(* IEC 61131-3 sources: CodesysTest/export/UN00 - Sharp Bagger/EM01 - Bagger Head/CM04 - Bag Delivery/FB_SXBagDelivery.pou, 3 files *)

(* ---- FB_SXBagDelivery.pou.st ---- *)
(*#-#-#-#-#-#-#-#-#-#---Declaration---#-#-#-#-#-#-#-#-#-#-#-#-#*)

FUNCTION_BLOCK FINAL FB_SXBagDelivery EXTENDS FB_BaseComponent IMPLEMENTS IBagDelivery
VAR_INPUT
	simulateIO : BOOL;
	dryCycleEnable : BOOL;
	bagPresent : BOOL;
	printer : IPrinter;
	bagLength : REAL := 24.0;
	feedSpeed : REAL := 30.0;
	reverseSpeed : REAL := 3.0;
	printSpeed : REAL := 6.0;
	printOffset : REAL := 4.5;
	printLength : REAL := 6.0;
	maxReverseSetpoint : REAL := 3.0;
	sealOffset : REAL := 1.5;
	distanceFromSealBarToBagEdge : REAL := 3;
	distanceFromNipToBagEdge : REAL := 1.25;
	trapezoidalPercent : REAL := 0.1;
END_VAR
VAR_OUTPUT
	reverseFault : FB_Fault(name := Standard.CONCAT(_prefix,'Reverse Fault'));
	bagFailedToSeparate : FB_Fault(name := Standard.CONCAT(_prefix,'Failed To Separate'));
	noBagOverEye : FB_Fault(name := Standard.CONCAT(_prefix,'No Bag Over Photoeye'));
	motorFault : FB_Fault(name := CONCAT(_prefix, 'Film Feed Motor Fault'));
	motorCommFault : FB_Fault(name := CONCAT(_prefix, 'Film Feed Motor Comm Fault'));
END_VAR
VAR
	_feedAtPrintSpeed : BOOL;
	_feedBagOut : BOOL;
	_feedToPrintOffset : BOOL;
	_reverseToSeparate : BOOL;
	_bagFeedDone : BOOL;
	_bagSeparated : BOOL;
	_readyForPrint : BOOL;
	state : INT;
	nextState : INT;
	moveBagDeliveryTimeout : Standard.TON;
	MC_MoveBagDelivery : MC_MoveRelative;
	MC_HaltBagDelivery : MC_Halt;
	MC_ResetBagDelivery : MC_Reset;
	remainingLength : REAL;
	bagReversedToPrintOffset : BOOL;
	bagEdgePhotoeyeSim : FB_SimulatedFeedbackPhysicalInput(name := 'Bag Edge Photoeye Sim');
	printingNow : BOOL;
END_VAR
VAR_IN_OUT
	bagDeliveryMotor : Axis_REF;
END_VAR(*#-#-#-#-#-#-#-#-#-#---Implementation---#-#-#-#-#-#-#-#-#-#-#-#-#*)

SUPER^();

{region "Axis Setup"}
// Setup of Motion Commands for Bag Delivery motor axis
MC_MoveBagDelivery(Axis := bagDeliveryMotor);
MC_HaltBagDelivery(Axis := bagDeliveryMotor);
MC_ResetBagDelivery(Axis := bagDeliveryMotor);
{endregion}

IF MC_ResetBagDelivery.Execute THEN
	MC_ResetBagDelivery.Execute := FALSE;
END_IF

IF resetONS.Q THEN
	state := 100;
	nextState := 0;
	ClearStatus();
	IF bagDeliveryMotor.Error OR NOT bagDeliveryMotor.CommStatus THEN
		MC_ResetBagDelivery.Execute := TRUE;
	END_IF
END_IF

_ready := state = 0 AND bagDeliveryMotor.CommStatus AND NOT bagDeliveryMotor.Error;
IF bagDeliveryMotor.Error THEN
	motorFault.faultTrigger := TRUE;
ELSE
	motorFault.faultTrigger := FALSE;
END_IF

IF NOT bagDeliveryMotor.CommStatus THEN
	motorCommFault.faultTrigger := TRUE;
ELSE
	motorCommFault.faultTrigger := FALSE;
END_IF

IF trapezoidalPercent <= 0 THEN
	trapezoidalPercent := 0.1;
END_IF

CASE state OF
	0:		// Idle
			IF _feedBagOut THEN
				state := 10;
				_feedBagOut := FALSE;
				ClearStatus();
			END_IF

			IF _feedToPrintOffset THEN
				state := 20;
				_feedToPrintOffset := FALSE;
				ClearStatus();
			END_IF

			IF _reverseToSeparate THEN
				_bagSeparated := FALSE;
				state := 50;
				_reverseToSeparate := FALSE;
				ClearStatus();
			END_IF

			IF _feedAtPrintSpeed THEN
				state := 40;
				_feedAtPrintSpeed := FALSE;
				ClearStatus();
			END_IF

	1:		// Homing

	2:		//

	4: 		//

	5:		//

	6:		//

	7:		//

	10:		// Feed bag out
			MC_MoveBagDelivery.Acceleration := MC_MoveBagDelivery.Deceleration := (feedSpeed / trapezoidalPercent);
			MC_MoveBagDelivery.Velocity := feedSpeed;
			MC_MoveBagDelivery.Distance := remainingLength;
			moveBagDeliveryTimeout.PT := MoveTimeoutCalc(remainingLength, feedSpeed, 1000);
			moveBagDeliveryTimeout.IN := TRUE;
			MC_MoveBagDelivery.Execute := TRUE;
			_logger.AddLogItem(CONCAT(_prefix, 'Feeding Bag Out'));
			state := 101;
			nextState := 11;

	11:		// Set Bag Feed Done
			_bagFeedDone := TRUE;
			_logger.AddLogItem(CONCAT(_prefix, 'Bag Feed Done'));
			state := 0;
			nextState := 0;

	20:		// Feed bag to print offset.  If already at print offset from reversing, continue
			IF bagReversedToPrintOffset THEN
				state := 21;
				nextState := 0;
				bagReversedToPrintOffset := FALSE;
			ELSE
				MC_MoveBagDelivery.Acceleration := MC_MoveBagDelivery.Deceleration := (feedSpeed / trapezoidalPercent);
				MC_MoveBagDelivery.Velocity := feedSpeed;
				MC_MoveBagDelivery.Distance := printOffset;
				remainingLength := remainingLength - printOffset;
				moveBagDeliveryTimeout.PT := MoveTimeoutCalc(printOffset, feedSpeed, 1000);
				moveBagDeliveryTimeout.IN := TRUE;
				MC_MoveBagDelivery.Execute := TRUE;
				_logger.AddLogItem(CONCAT(_prefix, 'Feeding Bag to Print Offset'));

				state := 101;
				nextState := 21;
			END_IF

	21: 	// Set Ready For Print
			_readyForPrint := TRUE;
			state := 0;
			nextState := 0;

	50: 	// Feed bag if not over photoeye
			IF NOT bagPresent AND NOT dryCycleEnable THEN
				MC_MoveBagDelivery.Acceleration := MC_MoveBagDelivery.Deceleration := (reverseSpeed / trapezoidalPercent);
				MC_MoveBagDelivery.Velocity := reverseSpeed;
				MC_MoveBagDelivery.Distance := maxReverseSetpoint;
				moveBagDeliveryTimeout.PT := MoveTimeoutCalc(maxReverseSetpoint, reverseSpeed, 1000);
				moveBagDeliveryTimeout.IN := TRUE;
				MC_MoveBagDelivery.Execute := TRUE;
				_logger.AddLogItem(CONCAT(_prefix, 'Feed to Photoeye'));
				//bagEdgePhotoeyeSim.in := TRUE;
				state := 51;
			ELSE
				state := 30;
			END_IF

	51: 	// If move completed then fault, otherwise stop at photoeye
			IF MC_MoveBagDelivery.Done THEN
				MC_MoveBagDelivery.Execute := FALSE;
				noBagOverEye.Trigger();
				ClearStatus();
				state := 100;
				nextState := 0;
			END_IF

			IF MC_MoveBagDelivery.Error OR moveBagDeliveryTimeout.Q THEN
				reverseFault.Trigger();
				MC_MoveBagDelivery.Execute := FALSE;
				MC_HaltBagDelivery.Execute := TRUE;
				ClearStatus();
				nextState := 0;
				state := 100;
			END_IF

			IF bagPresent THEN
				MC_MoveBagDelivery.Execute := FALSE;
				MC_HaltBagDelivery.Execute := TRUE;
				bagEdgePhotoeyeSim.in := FALSE;
				state := 52;

			END_IF

	52:		// Wait for bag to stop
			IF MC_HaltBagDelivery.Done THEN
				MC_HaltBagDelivery.Execute := FALSE;
				state := 30;
			END_IF

	30:		// Reverse to Separate
			MC_MoveBagDelivery.Acceleration := MC_MoveBagDelivery.Deceleration := (reverseSpeed / trapezoidalPercent);
			MC_MoveBagDelivery.Velocity := reverseSpeed;
			MC_MoveBagDelivery.Distance := maxReverseSetpoint * -1;
			moveBagDeliveryTimeout.PT := MoveTimeoutCalc(maxReverseSetpoint, reverseSpeed, 1000);
			moveBagDeliveryTimeout.IN := TRUE;
			MC_MoveBagDelivery.Execute := TRUE;
			_logger.AddLogItem(CONCAT(_prefix, 'Reversing to Photoeye'));
			bagEdgePhotoeyeSim.in := TRUE;
			state := 31;
			//nextState := 31;

	31:		// Stop bag once edge clears photoeye. If move command finishes that means the bag didn't separate
			IF MC_MoveBagDelivery.Done AND NOT dryCycleEnable THEN
				MC_MoveBagDelivery.Execute := FALSE;
				bagFailedToSeparate.Trigger();
				ClearStatus();
				state := 100;
				nextState := 0;
			END_IF

			IF MC_MoveBagDelivery.Done AND dryCycleEnable THEN
				MC_MoveBagDelivery.Execute := FALSE;
				MC_HaltBagDelivery.Execute := FALSE;
				bagEdgePhotoeyeSim.in := FALSE;
				state := 32;
			END_IF

			IF MC_MoveBagDelivery.Error OR moveBagDeliveryTimeout.Q THEN
				reverseFault.Trigger();
				MC_MoveBagDelivery.Execute := FALSE;
				MC_HaltBagDelivery.Execute := TRUE;
				ClearStatus();
				nextState := 32;
				state := 100;
			END_IF

			IF NOT bagPresent AND NOT dryCycleEnable THEN
				MC_MoveBagDelivery.Execute := FALSE;
				MC_HaltBagDelivery.Execute := TRUE;
				bagEdgePhotoeyeSim.in := FALSE;
				state := 32;
			END_IF

	32: 	// Set Bag Reversed
			IF MC_HaltBagDelivery.Done OR dryCycleEnable THEN
				MC_HaltBagDelivery.Execute := FALSE;
				remainingLength := bagLength - sealOffset + distanceFromSealBarToBagEdge;
				_bagSeparated := TRUE;
				state := 0;
				nextState := 0;
			END_IF

	40:		// Feed at Print Speed
			MC_MoveBagDelivery.Acceleration := MC_MoveBagDelivery.Deceleration := (printSpeed / trapezoidalPercent);
			MC_MoveBagDelivery.Velocity := printSpeed;
			MC_MoveBagDelivery.Distance := printLength;
			moveBagDeliveryTimeout.PT := MoveTimeoutCalc(distanceFromNipToBagEdge, reverseSpeed, 1000);
			moveBagDeliveryTimeout.IN := TRUE;
			MC_MoveBagDelivery.Execute := TRUE;
			_logger.AddLogItem(CONCAT(_prefix, 'Feeding At Print Speed'));
			remainingLength := remainingLength - printLength;
			_feedBagOut := FALSE;
			printingNow := TRUE;
			state := 101;
			nextState := 10;

	100:	// Cleanup
			MC_MoveBagDelivery.Execute := FALSE;
			MC_HaltBagDelivery.Execute := FALSE;
			moveBagDeliveryTimeout.IN := FALSE;
			bagEdgePhotoeyeSim.in := FALSE;
			state := nextState;

	101: 	// Wait for Move to complete
			IF MC_MoveBagDelivery.Error OR moveBagDeliveryTimeout.Q THEN
				MC_MoveBagDelivery.Execute := FALSE;
				MC_HaltBagDelivery.Execute := TRUE;
				ClearStatus();
				nextState := 0;
				state := 100;
			END_IF

			IF MC_MoveBagDelivery.Done THEN
				IF printingNow THEN
					printer.StopPrinting();
					IF printer.PrintDone THEN
						printingNow := FALSE;
						moveBagDeliveryTimeout.IN := FALSE;
						MC_MoveBagDelivery.Execute := FALSE;
						state := nextState;
					END_IF
				ELSE
					moveBagDeliveryTimeout.IN := FALSE;
					MC_MoveBagDelivery.Execute := FALSE;
					state := nextState;
				END_IF
			END_IF

	103:	// Set In Position and go back to idle
			nextState := 0;
			state := 100;

END_CASE

(* ---- ClearStatus.m.st ---- *)
(*#-#-#-#-#-#-#-#-#-#---Declaration---#-#-#-#-#-#-#-#-#-#-#-#-#*)

METHOD ClearStatus
VAR_INPUT
END_VAR
(*#-#-#-#-#-#-#-#-#-#---Implementation---#-#-#-#-#-#-#-#-#-#-#-#-#*)

_bagFeedDone := FALSE;
_bagSeparated := FALSE;
_readyForPrint := FALSE;
printingNow := FALSE;

(* ---- FeedToPhotoeye.m.st ---- *)
(*#-#-#-#-#-#-#-#-#-#---Declaration---#-#-#-#-#-#-#-#-#-#-#-#-#*)

METHOD FeedToPhotoeye
VAR_INPUT
END_VAR(*#-#-#-#-#-#-#-#-#-#---Implementation---#-#-#-#-#-#-#-#-#-#-#-#-#*)
